% RSLogix 500 project Batch Mixing Process.RSS, saved by version 8.30.01.01 %
PROJECT "UNTITLED"    % processor: Bul.1763 MicroLogix 1100 Series B %

PROGRAM FILES
  LAD 2   7 rungs

DATA FILES
  O0 OUTPUT  4 elements
  I1 INPUT  6 elements
  S2 STATUS  66 elements
  B3 BINARY  1 elements
  T4 TIMER  1 elements
  C5 COUNTER  2 elements
  R6 CONTROL  1 elements
  N7 INTEGER  1 elements
  F8 FLOAT  1 elements

LADDER 2
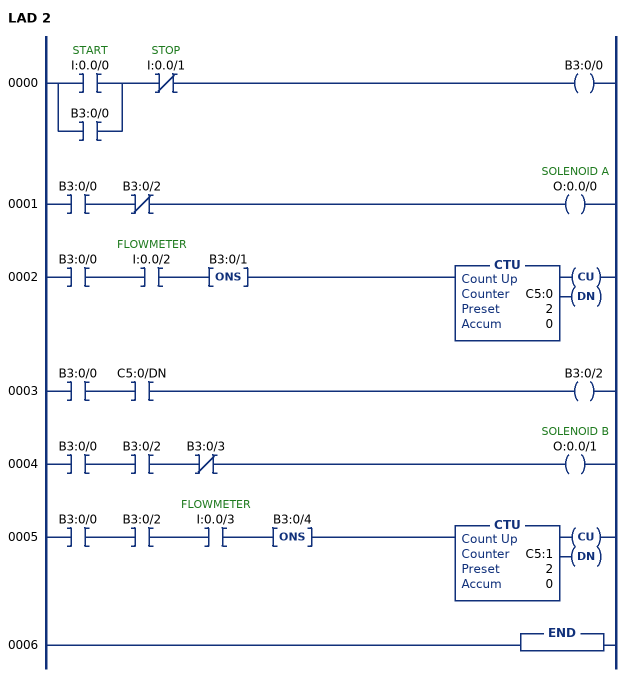
% Rung: 0 %  % edit flag set %
SOR BST XIC I:0.0/0 NXB XIC B3:0/0 BND XIO I:0.0/1 OTE B3:0/0 EOR
%   I:0.0/0  "START" %
%   I:0.0/1  "STOP" %
% Rung: 1 %  % edit flag set %
SOR XIC B3:0/0 XIO B3:0/2 OTE O:0.0/0 EOR
%   O:0.0/0  "SOLENOID A" %
% Rung: 2 %  % edit flag set %
SOR XIC B3:0/0 XIC I:0.0/2 ONS B3:0/1 CTU C5:0 2 0 EOR
%   I:0.0/2  "FLOWMETER" %
% Rung: 3 %  % edit flag set %
SOR XIC B3:0/0 XIC C5:0/DN OTE B3:0/2 EOR
% Rung: 4 %  % edit flag set %
SOR XIC B3:0/0 XIC B3:0/2 XIO B3:0/3 OTE O:0.0/1 EOR
%   O:0.0/1  "SOLENOID B" %
% Rung: 5 %  % edit flag set %
SOR XIC B3:0/0 XIC B3:0/2 XIC I:0.0/3 ONS B3:0/4 CTU C5:1 2 0 EOR
%   I:0.0/3  "FLOWMETER" %
% Rung: 6 %
SOR END EOR
